{attribute 'qualified_only'}
{attribute 'strict'}
{attribute 'to_string'}
TYPE E_MESSAGE_CTRL :
(
	MSG_CTRL_NULL,
	MSG_CTRL_INIT   := 10,
  MSG_CTRL_IDLE   := 30,
  MSG_CTRL_WRITE  := 50
)UINT;
END_TYPE

(* stored: Version 1.1.0.1
   DUT E_MESSAGE_CTRL: Id {9c313f81-5e95-4dd0-9e6e-b83be0ac707b} *)
